PROGRAM MAIN
VAR
	estate 			: 	E_TestState := E_TestState.IDLE;	// different test states for the functions
	lat, lon        :   LREAL;							// location for observer						
	ra, dec			:   LREAL;							// coord eq
	alt, az			:   LREAL;							// coord eq
	eq2hor			:	FB_EQ2HOR;						// equatorial to horizontal transform function block (Stella1) (J2000) in degrees (FK5)
	hor2eq			:	FB_HOR2EQ;						// horizontal to equatorial transform function block (Stella1) (J2000) in degrees (FK5)
	
	lst1			: 	LREAL;
	jd1				:	LREAL;
	cycle_time		:	LREAL;
END_VAR

CASE estate OF
	E_TestState.IDLE:
		estate := E_TestState.IDLE;
		
		
	E_TestState.JD2LST:
		// transform time
		lst1 := JD2LST(jd := jd1, lon := lon, dut1 := 0.0);
		// return to IDLE
		cycle_time := UDINT_TO_LREAL(_TaskInfo[GETCURTASKINDEXEX()].CycleTime) / 10_000_000;
		estate := E_TestState.IDLE;
		
		
	E_TestState.EQ2HOR:
		// transform coordinates
		eq2hor(ra:=ra, dec:=dec, jd:=jd1, lon:=lon, lat:=lat, refract:=FALSE, alt=>alt, az=>az);
		// return to IDLE
		cycle_time := UDINT_TO_LREAL(_TaskInfo[GETCURTASKINDEXEX()].CycleTime) / 10_000_000;
		estate := E_TestState.IDLE;
	E_TestState.EQ2EQ:
		// transform to ALT AZ
		eq2hor(ra:=ra, dec:=dec, JD:=jd1, lon:=lon, lat:=lat, refract:=FALSE, alt=>alt, az=>az);
		// transform back :)
		hor2eq(alt:=alt, az:=az, jd:=jd1,lon:=lon, lat:=lat, refract:=FALSE, ra=>ra, dec=>dec);
		estate := E_TestState.IDLE;
	E_TestState.HOR2EQ:
		// transform :)
		hor2eq(alt:=alt, az:=az, jd:=jd1 , lon:=lon, lat:=lat, refract:=FALSE, ra=>ra, dec=>dec);
		estate := E_TestState.IDLE;
END_CASE

END_PROGRAM

(* stored: Version 1.1.0.1, ProductVersion 3.1.4024.12
   POU MAIN: Id {9edd3dc7-464a-45b7-b5f9-e2076842766b}, SpecialFunc None *)
